FUNCTION_BLOCK T_ModuleCollectionSetSubModuleInfoActiveSuccess EXTENDS T_UnitTestBase
VAR
  list : T_SubModuleCollection(10);
  newModule, newModule2 : T_SubModuleMock; 
  actual1, actual2, result : BOOL;

  PMLSubModuleInfo  : ARRAY[1..10] OF ST_PMLSubUnitInfo;
END_VAR

// Arrange
list.AddModule(newModule);
list.AddModule(newModule2);

//Act
result := list.SetPMLSubModuleInfoActive(PMLSubModuleInfo);

//Assert
actual1:=  PMLSubModuleInfo[1].Active;
actual2:=  PMLSubModuleInfo[2].Active;

assertion.AssertEquals_BOOL(TRUE, actual1, 'actual1:=  PMLSubModuleInfo[1].Active;');
assertion.AssertEquals_BOOL(TRUE, actual2, 'actual2:=  PMLSubModuleInfo[2].Active;');
assertion.AssertEquals_BOOL(TRUE, result, 'result := list.SetPMLSubModuleInfoActive(PMLSubModuleInfo);');
TestFinished();

END_FUNCTION_BLOCK

(* stored: Version 1.1.0.1, ProductVersion 3.1.4024.12
   POU T_ModuleCollectionSetSubModuleInfoActiveSuccess: Id {a7baad53-ced4-4e4e-b17f-06e0652e042c}, SpecialFunc None *)
